// TIA Portal V17 export
// export: Created 2024-08-26T21:07:19.8283581Z, ExportSetting WithDefaults, DisplayName Totally Integrated Automation Portal, DisplayVersion V17 Update 7, DisplayName TIA Portal Openness, DisplayVersion V17 Update 7, DisplayName TIA Portal Version Control Interface, DisplayVersion V17, DisplayName SINAMICS Startdrive Advanced, DisplayVersion V17 SP2, DisplayName SINAMICS Startdrive G110M, G120, G120C, G120D, G120P, G115D, DisplayVersion V17 SP2, DisplayName SINAMICS Startdrive G130, G150, S120, S150, SINAMICS MV, S210, DisplayVersion V17 SP2, DisplayName STEP 7 Professional, DisplayVersion V17 Update 7, DisplayName STEP 7 Safety, DisplayVersion V17 Update 6, DisplayName WinCC Advanced / Unified PC, DisplayVersion V17 Update 7
DATA_BLOCK "DB_INST_AWAKE_SIGNAL"   // DB1003
VERSION : 0.1
// stored: AutoNumber false, DBAccessibleFromOPCUA true, DBAccessibleFromWebserver true, InstanceOfName FB_IJC_AWAKE_SIGNAL, InstanceOfType FB
"FB_IJC_AWAKE_SIGNAL"
   // VAR_INPUT
   //    ack_error : Bool;
   // END_VAR
   // VAR_OUTPUT
   //    State_com : SInt;
   // END_VAR
   // VAR
   //    T1PresetValue : Time;
   //    T2PresetValue : Time;
   //    AwSignalTimeOutFault : Bool;
   //    Reset_Counters : Bool;
   //    Restart_Counter_bit_of_life : USInt;
   //    NB_Bit_of_Life : Bool;
   //    number_restart : DInt;
   //    check_restart : Bool;
   //    "Timer" { ExternalAccessible := 'False'; ExternalVisible := 'False'; ExternalWritable := 'False'} : Array[1..5] of TON_TIME;
   // END_VAR
BEGIN
END_DATA_BLOCK
